// TIA Portal project "kamery funkcni_V13_SP1_V14" (V14)

(* hardware
DEVICE "SIMATIC 1200 station_1"  S71200.Device
   slot 0: "S7-1200 rack"  Rack  V1.0
   slot 1: "PLC_1"  CPU 1214C DC/DC/DC  6ES7 214-1AG31-0XB0  V3.0
DEVICE "HMI_1"  KTP400 Basic color PN
   slot 0: "HMI"  HMI  6AV6 647-0AK11-3AX0  11.0.2
   slot 1: "HMI_RT_1"  KTP400 Basic PN  6AV6 647-0AK11-3AX0  11.0.2
   slot 5: "IE_CP_1"  PROFINET interface  IE_CP  V7.1.0
      slot 1: "PROFINET_Interface_1"  HMI IE SUBMODULE
         slot 1: "PORT_1"  HMI IE PORTMODULE 1  1.0.0.0
*)

// ===== PLC "PLC_1"  CPU 1214C DC/DC/DC =====

VAR_GLOBAL   // PLC tag table "Default tag table"
   "Tag_1" AT %MB12 : Byte;
   "Tag_2" AT %QB0 : Byte;
   "SEND" AT %M10.0 : Bool;
   "Clock_Byte" AT %MB0 : Byte;
   "Clock_10Hz" AT %M0.0 : Bool;
   "Clock_5Hz" AT %M0.1 : Bool;
   "Clock_2.5Hz" AT %M0.2 : Bool;
   "Clock_2Hz" AT %M0.3 : Bool;
   "Clock_1.25Hz" AT %M0.4 : Bool;
   "Clock_1Hz" AT %M0.5 : Bool;
   "Clock_0.625Hz" AT %M0.6 : Bool;
   "Clock_0.5Hz" AT %M0.7 : Bool;
   "System_Byte" AT %MB1 : Byte;
   "FirstScan" AT %M1.0 : Bool;
   "DiagStatusUpdate" AT %M1.1 : Bool;
   "AlwaysTRUE" AT %M1.2 : Bool;
   "AlwaysFALSE" AT %M1.3 : Bool;
END_VAR

DATA_BLOCK "Data_block_1"   // DB3
{ S7_Optimized_Access := 'TRUE' }
VERSION : 0.1
   VAR
      DATA_RCV : String;
      DATA_SEND : String;
      DATA_RCV_ARRAY : Array[0..12] of Char;
      dIS : String;
   END_VAR
BEGIN
END_DATA_BLOCK

// folder: System blocks/Program resources

DATA_BLOCK "PLC_1_Receive_DB"   // DB2
{ S7_Optimized_Access := 'TRUE' }
AUTHOR : SIMATIC
FAMILY : MC7Plus
NAME : TCON_Prm
VERSION : 1.0
// stored: InstanceOfName TCON_Param
"TCON_Param"
BEGIN
   ID := 5;
   ACTIVE_EST := false;
   REM_TSAP_ID_LEN := 0;
   LOCAL_TSAP_ID[1] := B#16#07;
   LOCAL_TSAP_ID[2] := B#16#D0;
   LOCAL_TSAP_ID_LEN := 2;
   REM_STADDR_LEN := 0;
END_DATA_BLOCK

DATA_BLOCK "IEC_Timer_0_DB"   // DB5
{ S7_Optimized_Access := 'TRUE' }
AUTHOR : Simatic
FAMILY : IEC
NAME : IEC_TMR
VERSION : 1.0
// stored: InstanceOfName IEC_TIMER
"IEC_TIMER"
BEGIN
END_DATA_BLOCK

DATA_BLOCK "PLC_1_Send_DB"   // DB6
{ S7_Optimized_Access := 'TRUE' }
AUTHOR : SIMATIC
FAMILY : MC7Plus
NAME : TCON_Prm
VERSION : 1.0
// stored: InstanceOfName TCON_Param
"TCON_Param"
BEGIN
   ID := 1;
   REM_TSAP_ID[1] := B#16#11;
   REM_TSAP_ID[2] := B#16#46;
   LOCAL_TSAP_ID[1] := B#16#07;
   LOCAL_TSAP_ID[2] := B#16#D1;
   LOCAL_TSAP_ID_LEN := 2;
   REM_STADDR[1] := 192;
   REM_STADDR[2] := 168;
   REM_STADDR[3] := 1;
   REM_STADDR[4] := 100;
END_DATA_BLOCK

DATA_BLOCK "PLC_1_Connection_DB"   // DB7
{ S7_Optimized_Access := 'TRUE' }
AUTHOR : SIMATIC
FAMILY : MC7Plus
NAME : TCON_Prm
VERSION : 1.0
// stored: InstanceOfName TCON_Param
"TCON_Param"
BEGIN
   ID := 2;
   REM_TSAP_ID[1] := B#16#07;
   REM_TSAP_ID[2] := B#16#D0;
   REM_STADDR[1] := 192;
   REM_STADDR[2] := 168;
   REM_STADDR[3] := 1;
   REM_STADDR[4] := 191;
END_DATA_BLOCK

DATA_BLOCK "PLC_1_Connection_DB_1"   // DB8
{ S7_Optimized_Access := 'TRUE' }
AUTHOR : SIMATIC
FAMILY : MC7Plus
NAME : TCON_Prm
VERSION : 1.0
// stored: InstanceOfName TCON_Param
"TCON_Param"
BEGIN
   ID := 4;
   REM_TSAP_ID[1] := B#16#07;
   REM_TSAP_ID[2] := B#16#D0;
   REM_STADDR[1] := 192;
   REM_STADDR[2] := 168;
   REM_STADDR[3] := 1;
   REM_STADDR[4] := 191;
END_DATA_BLOCK

// folder: (top level)

ORGANIZATION_BLOCK "Main"   // OB1, LAD, ProgramCycle
TITLE = "Main Program Sweep (Cycle)"
{ S7_Optimized_Access := 'TRUE' }
VERSION : 0.1
BEGIN

REGION Network 1
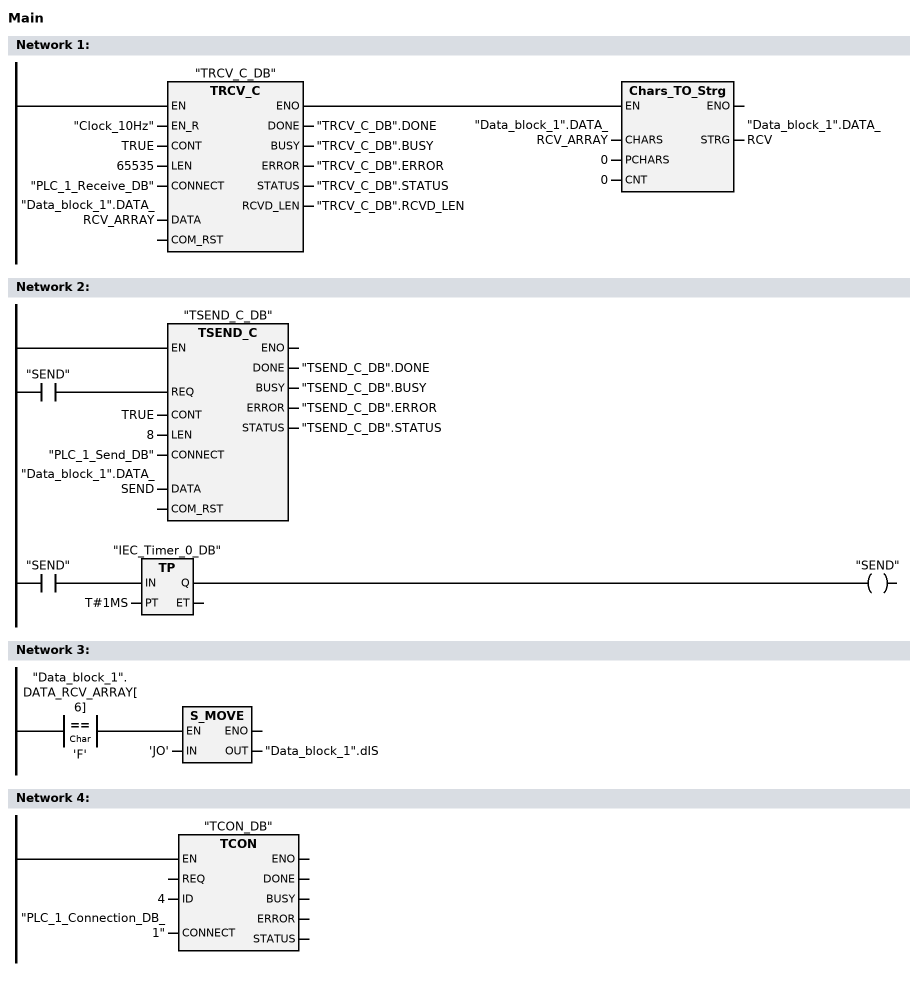
   // no SCL statement known for Chars_TO_Strg: written as a call
   // ENO of a box is taken as its EN; it also drops when the box reports an error
   "TRCV_C_DB"(EN_R := "Clock_10Hz",   // TRCV_C
               CONT := TRUE,
               LEN := 65535,
               CONNECT := "PLC_1_Receive_DB",
               DATA := "Data_block_1".DATA_RCV_ARRAY,
               DONE => "TRCV_C_DB".DONE,
               BUSY => "TRCV_C_DB".BUSY,
               ERROR => "TRCV_C_DB".ERROR,
               STATUS => "TRCV_C_DB".STATUS,
               RCVD_LEN => "TRCV_C_DB".RCVD_LEN);
   Chars_TO_Strg(Chars := "Data_block_1".DATA_RCV_ARRAY, pChars := 0, Cnt := 0, Strg => "Data_block_1".DATA_RCV);
END_REGION

REGION Network 2
   "TSEND_C_DB"(REQ := "SEND",   // TSEND_C
                CONT := TRUE,
                LEN := 8,
                CONNECT := "PLC_1_Send_DB",
                DATA := "Data_block_1".DATA_SEND,
                DONE => "TSEND_C_DB".DONE,
                BUSY => "TSEND_C_DB".BUSY,
                ERROR => "TSEND_C_DB".ERROR,
                STATUS => "TSEND_C_DB".STATUS);
   "IEC_Timer_0_DB".TP(IN := "SEND", PT := T#1MS);
   "SEND" := "IEC_Timer_0_DB".Q;
END_REGION

REGION Network 3
   RUNG wire#powerrail
      { S7_Templates := "SrcType := Char" } EQ_Contact(in1 := "Data_block_1".DATA_RCV_ARRAY[6], in2 := 'F')
      { S7_GenerateENO := "TRUE" } S_Move(in := 'JO', out => "Data_block_1".dIS)
   END_RUNG
   // the same network as SCL:
   IF "Data_block_1".DATA_RCV_ARRAY[6] = 'F' THEN "Data_block_1".dIS := 'JO'; END_IF;
END_REGION

REGION Network 4
   "TCON_DB"(ID := 4, CONNECT := "PLC_1_Connection_DB_1");   // TCON
END_REGION
END_ORGANIZATION_BLOCK

(* ===== HMI "HMI_RT_1" =====
system functions are stored by id; their names below are inferred from use
connection "HMI_connection": ETHERNET, SMART_S7_1200

HMI tags "Default tag table"
   "Data_block_1_DATA_RCV" : String[254] = PLC Data_block_1.DATA_RCV, 100 ms
   "SEND" : Bool = PLC SEND AT %M10.0, 100 ms
   "Data_block_1_DATA_SEND" : String[254] = PLC Data_block_1.DATA_SEND, 100 ms
   "Data_block_1_dIS" : String[254] = PLC Data_block_1.dIS, 1 s

text list "Text_list_1": 0 ''

screen "Root screen" 480x272, template "Template_1"
   Button "Button_1" at 145,123 size 112x55; TextOff 'SEND'
      on Click: SetTag("SEND", 1)
   IOField "I/O field_1" at 290,135 size 188x35; FormatPattern ?????????????
      ProcessValue <- "Data_block_1_DATA_RCV"
   IOField "I/O field_2" at 15,138 size 112x32; FormatPattern ??????
      ProcessValue <- "Data_block_1_DATA_SEND"
   TextField "Text field_1" at 290,106 size 106x20; Text 'Odezva kamery'
   TextField "Text field_2" at 15,106 size 114x20; Text 'Vstup do kamery'
   IOField "I/O field_3" at 307,31 size 90x32; FormatPattern ??????????
      ProcessValue <- "Data_block_1_dIS"
*)